PROGRAM MAIN
VAR
END_VAR

PLC_Mode() ;

SQL_Mode();

END_PROGRAM

(* stored: Version 1.1.0.1, ProductVersion 3.1.4024.12
   POU MAIN: Id {cda6c0d4-7565-48ec-9eb7-3c245b63c961}, SpecialFunc None *)
